// TIA Portal V17 export
// export: Created 2024-09-02T12:50:28.8021989Z, ExportSetting WithDefaults, DisplayName Totally Integrated Automation Portal, DisplayVersion V17, DisplayName TIA Portal Openness, DisplayVersion V17, DisplayName TIA Portal Version Control Interface, DisplayVersion V17, DisplayName STEP 7 Professional, DisplayVersion V17, DisplayName STEP 7 Safety, DisplayVersion V17, DisplayName WinCC Professional, DisplayVersion V17
TYPE "TypeSKS_OPERATOR"
// stored: IsFailsafeCompliant false
   STRUCT
      BEA { ExternalWritable := 'False'} : Array[1..8] of Struct
         permission { ExternalWritable := 'False'} : Bool;
         ok { ExternalWritable := 'False'} : Bool;
         nok { ExternalWritable := 'False'} : Bool;
         "repeat" { ExternalWritable := 'False'} : Bool;
      END_STRUCT;
   END_STRUCT;
END_TYPE
